// Layout checklist: STRING(n) and WSTRING(n) sizes.
// The guard byte behind the narrow string shows whether the terminator is
// counted; the wide string's own offset shows whether it is WORD-aligned,
// and the trailing byte whether that alignment pads the type out.
TYPE ST_StringSizes :
STRUCT
	narrow : STRING(5);
	guard : BYTE;
	wide : WSTRING(5);
	trailer : BYTE;
END_STRUCT
END_TYPE

(* stored: Version 1.1.0.1, ProductVersion 3.1.4026.18
   DUT ST_StringSizes: Id {c0de1a70-0000-4000-8000-000000000008} *)
